(* IEC 61131-3 sources: CodesysTest/alpha/export/Device.dev/Plc Logic/Application/FBs/Fault/FB_Fault.pou, 2 files *)

(* ---- Ack.m.st ---- *)
(*#-#-#-#-#-#-#-#-#-#---Declaration---#-#-#-#-#-#-#-#-#-#-#-#-#*)

METHOD Ack(*#-#-#-#-#-#-#-#-#-#---Implementation---#-#-#-#-#-#-#-#-#-#-#-#-#*)

IF _ackCommand OR _acked THEN
	RETURN;
END_IF
_acked := TRUE;
// Log the ACK.
_logger.AddLogItem(CONCAT(InstanceName,  ' Acked'));

(* ---- RegisterLogger.m.st ---- *)
(*#-#-#-#-#-#-#-#-#-#---Declaration---#-#-#-#-#-#-#-#-#-#-#-#-#*)

METHOD RegisterLogger
VAR_INPUT
	internalLogger : IMachineLogger;
END_VAR
(*#-#-#-#-#-#-#-#-#-#---Implementation---#-#-#-#-#-#-#-#-#-#-#-#-#*)

_logger := internalLogger;
